FUNCTION "WL_4ByteToDint" : DInt
{ S7_Optimized_Access := 'TRUE' }
VERSION : 0.1
   VAR_INPUT
      Byte0 : Byte;
      Byte1 : Byte;
      Byte2 : Byte;
      Byte3 : Byte;
   END_VAR

   VAR_TEMP
      tempDword : DWord;
   END_VAR


BEGIN
	#tempDword.%B0 := #Byte0;
	#tempDword.%B1 := #Byte1;
	#tempDword.%B2 := #Byte2;
	#tempDword.%B3 := #Byte3;

	#WL_4ByteToDint := DWORD_TO_DINT(#tempDword);
END_FUNCTION

